# EPICS autosave request: iocBoot/sioc-li14-bl01/blen_manual.req
file "manual.req" AREA=LI14,POS=888,INST=BZ14888A
file "manual.req" AREA=LI14,POS=888,INST=BZ14888B
